{attribute 'GeneratedUsingTerminal: EL9930-0000-0016'}
{attribute addProperty BoxType "EL9930-0000-0016"}
{attribute addProperty Id "IO_InputsEMPTY_STRUCTURE0IO_OutputsEMPTY_STRUCTURE0WcStateAT %I*WcState_9091E0EB2InfoDataAT %I*InfoData_41C547A32"}
{attribute addProperty CRC "2805724723"}
{attribute addProperty Size "4"}
TYPE EL9930_A73BF633 EXTENDS EtcSlaveTerminalBase_947E5A46 :
STRUCT
	{attribute addProperty Name "IO_Inputs"}
	IO_Inputs : EMPTY_STRUCTURE;
	{attribute addProperty Name "IO_Outputs"}
	IO_Outputs : EMPTY_STRUCTURE;
	{attribute addProperty Name "WcState"}
	WcState : WcState_9091E0EB;
	{attribute addProperty Name "InfoData"}
	InfoData : InfoData_41C547A3;
END_STRUCT
END_TYPE

(* stored: Version 1.2.0.0, ProductVersion 3.1.4024.9
   DUT EL9930_A73BF633: Id {6565b375-7a24-4b91-9a8d-b477712a13d2} *)
